// TIA Portal project "7 Switches to Control Heater" (V17)
// 7 Switches to Control Heater
// PLC Example 26
// When Switch 1 and Switch 2 or Switch 3 and Switch 4 (pushbuttons) are turned ON (pressed) and then turned OFF (released), then Heater will be ON.
// When Switch 4 and Switch 5 or Switch 6 and Switch 7 (pushbuttons) are turned ON (pressed) and then turned OFF (released), then Heater will be OFF.

(* hardware
DEVICE "S7-1200 station_1"  S7-1200 Station
   slot 0: "Rack_0"  S7-1200 Rack  Rack  V1.0
   slot 1: "PLC_1"  CPU 1212C AC/DC/Rly  6ES7 212-1BE40-0XB0  V4.5
*)

// ===== PLC "PLC_1"  CPU 1212C AC/DC/Rly =====

VAR_GLOBAL   // PLC tag table "Default tag table"
   "PB" AT %I0.0 : Bool;
   "Switch 1" AT %I0.1 : Bool;
   "Switch 2" AT %I0.2 : Bool;
   "Switch 3" AT %I0.3 : Bool;
   "Switch 4" AT %I0.4 : Bool;
   "Switch 5" AT %I0.5 : Bool;
   "Switch 6" AT %I0.6 : Bool;
   "Switch 7" AT %I0.7 : Bool;
   "Heater" AT %Q0.0 : Bool;
   "Tag_1" AT %M0.0 : Bool;
   "Tag_2" AT %M0.1 : Bool;
END_VAR

ORGANIZATION_BLOCK "Main"   // OB1, LAD, ProgramCycle
TITLE = "Main Program Sweep (Cycle)"
{ S7_Optimized_Access := 'TRUE' }
VERSION : 0.1
   VAR_INPUT
      Initial_Call : Bool;   // Initial call of this OB
      Remanence : Bool;   // =True, if remanent data are available
   END_VAR
BEGIN

REGION Network 1
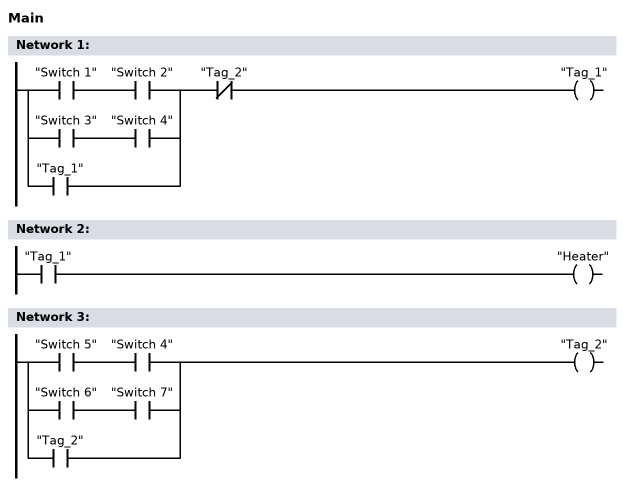
   RUNG wire#powerrail
      Contact( "Switch 1" )
      Contact( "Switch 2" )
      wire#w1
      I_Contact( "Tag_2" )
      Coil( "Tag_1" )
   END_RUNG
   RUNG wire#powerrail
      Contact( "Switch 3" )
      Contact( "Switch 4" )
   END_RUNG wire#w1
   RUNG wire#powerrail
      Contact( "Tag_1" )
   END_RUNG wire#w1
   // the same network as SCL:
   "Tag_1" := (("Switch 1" AND "Switch 2") OR ("Switch 3" AND "Switch 4") OR "Tag_1") AND NOT "Tag_2";
END_REGION

REGION Network 2
   RUNG wire#powerrail
      Contact( "Tag_1" )
      Coil( "Heater" )
   END_RUNG
   // the same network as SCL:
   "Heater" := "Tag_1";
END_REGION

REGION Network 3
   RUNG wire#powerrail
      Contact( "Switch 5" )
      Contact( "Switch 4" )
      wire#w1
      Coil( "Tag_2" )
   END_RUNG
   RUNG wire#powerrail
      Contact( "Switch 6" )
      Contact( "Switch 7" )
   END_RUNG wire#w1
   RUNG wire#powerrail
      Contact( "Tag_2" )
   END_RUNG wire#w1
   // the same network as SCL:
   "Tag_2" := ("Switch 5" AND "Switch 4") OR ("Switch 6" AND "Switch 7") OR "Tag_2";
END_REGION
END_ORGANIZATION_BLOCK